PROGRAM Safety
VAR
	uiEstopHandler : FB_HandleUiEstop;
	
	// Local variables
	_buttonPressed : BOOL;
	_resetPressed : BOOL;
	_stop : BOOL;
END_VAR


uiEstopHandler(
			button := _buttonPressed,
			reset := _resetPressed,
			stop => _stop);

PROPERTY buttonPressed : BOOL
SET

_buttonPressed := buttonPressed;
END_SET
END_PROPERTY

PROPERTY resetPressed : BOOL
SET

_resetPressed := resetPressed;
END_SET
END_PROPERTY

PROPERTY stop : BOOL
GET

stop := _stop;
END_GET
END_PROPERTY

END_PROGRAM

(* stored: Version 1.1.0.1, ProductVersion 3.1.4024.9
   POU Safety: Id {00b82d62-043d-415c-8b07-0526678ef84c}, SpecialFunc None
   Property buttonPressed: Id {d57cd45c-8045-45ca-af28-9cdd67208558}
   Set Set: Id {56101d58-a3ce-4e36-84d9-8c35a89552bc}
   Property resetPressed: Id {14ce5e0c-efc5-4e06-9c3e-b535b2438c4d}
   Set Set: Id {caed11da-48d4-4d5c-8e6c-97fb8799be26}
   Property stop: Id {347c660b-db44-463f-a2db-6e1c26aa510a}
   Get Get: Id {390803f4-119a-4c0f-af61-0772ee41a204} *)
